{attribute 'GeneratedUsingTerminal: EJ9576-0000-0022'}
{attribute addProperty BoxType "EJ9576-0000-0022"}
{attribute addProperty Id "EtcSlaveTerminalBaseBCT_InputsAT %I*BCT_Inputs_7ACE8FA617WcStateAT %I*WcState_9091E0EB2InfoDataAT %I*InfoData_32EB74EA10"}
{attribute addProperty CRC "3322871599"}
{attribute addProperty Size "29"}
TYPE EJ9576_C60EFF2F EXTENDS EtcSlaveTerminalBase :
STRUCT
	{attribute addProperty Name "BCT_Inputs"}
	BCT_Inputs : BCT_Inputs_7ACE8FA6;
	{attribute addProperty Name "WcState"}
	WcState : WcState_9091E0EB;
	{attribute addProperty Name "InfoData"}
	InfoData : InfoData_32EB74EA;
END_STRUCT
END_TYPE

(* stored: Version 1.2.0.0, ProductVersion 3.1.4024.9
   DUT EJ9576_C60EFF2F: Id {af1b040b-6f36-466b-888e-8f78c157479b} *)
